FUNCTION_BLOCK ResetPlotter (* Composite Function Block Type *)
  (* Standard: 61499-2 *)
  (* Version 1.0, 2020-03-02, Mario *)
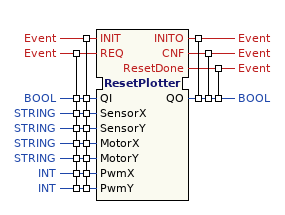
  EVENT_INPUT
    INIT WITH QI, SensorX, SensorY, MotorX, MotorY, PwmX, PwmY; (* Initialization Request *)
    REQ WITH QI, SensorX, SensorY, MotorX, MotorY, PwmX, PwmY; (* Normal Execution Request *)
  END_EVENT
  EVENT_OUTPUT
    INITO WITH QO; (* Initialization Confirm *)
    CNF WITH QO; (* Execution Confirmation *)
    ResetDone WITH QO;
  END_EVENT
  VAR_INPUT
    QI : BOOL; (* Input event qualifier *)
    SensorX : STRING;
    SensorY : STRING;
    MotorX : STRING;
    MotorY : STRING;
    PwmX : INT;
    PwmY : INT;
  END_VAR
  VAR_OUTPUT
    QO : BOOL; (* Output event qualifier *)
  END_VAR
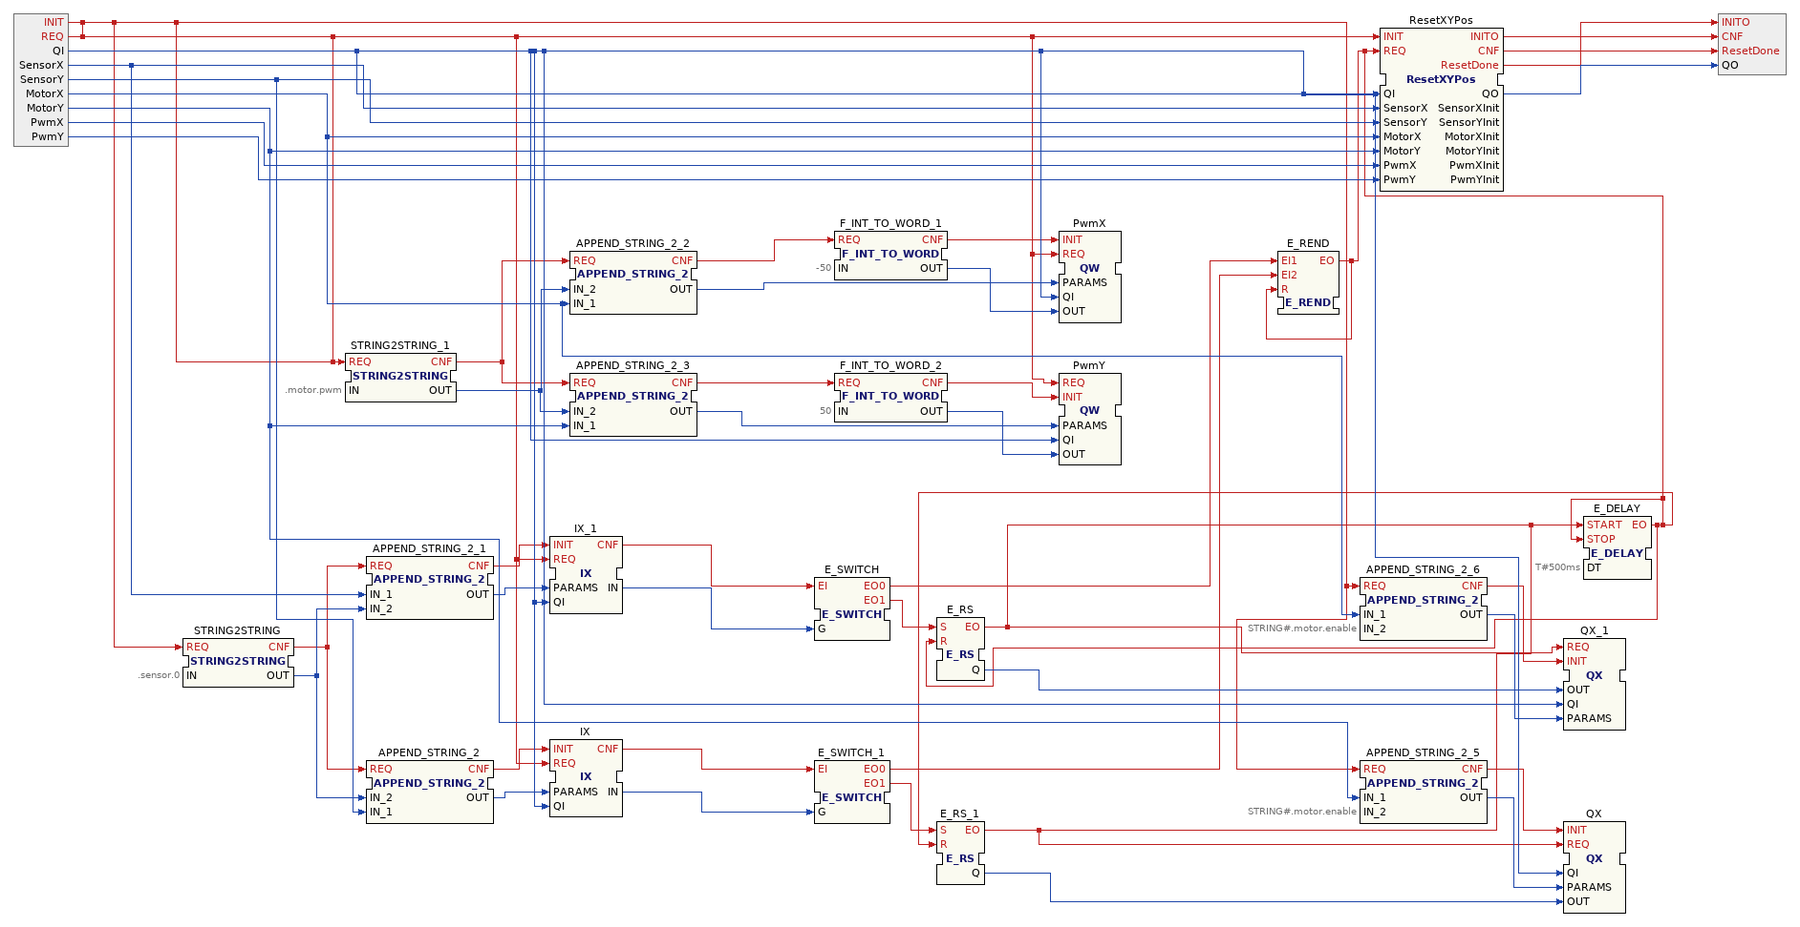
  FBS
    ResetXYPos : ResetXYPos;
    IX : IX;
    STRING2STRING : STRING2STRING(IN := .sensor.0);
    APPEND_STRING_2 : APPEND_STRING_2;
    IX_1 : IX;
    APPEND_STRING_2_1 : APPEND_STRING_2;
    E_SWITCH : E_SWITCH;
    E_SWITCH_1 : E_SWITCH;
    E_REND : E_REND;
    QX : QX;
    E_RS : E_RS;
    E_DELAY : E_DELAY(DT := T#500ms);
    PwmX : QW;
    PwmY : QW;
    STRING2STRING_1 : STRING2STRING(IN := .motor.pwm);
    APPEND_STRING_2_2 : APPEND_STRING_2;
    APPEND_STRING_2_3 : APPEND_STRING_2;
    QX_1 : QX;
    APPEND_STRING_2_5 : APPEND_STRING_2(IN_2 := STRING#.motor.enable);
    APPEND_STRING_2_6 : APPEND_STRING_2(IN_2 := STRING#.motor.enable);
    E_RS_1 : E_RS;
    F_INT_TO_WORD_1 : F_INT_TO_WORD(IN := -50);
    F_INT_TO_WORD_2 : F_INT_TO_WORD(IN := 50);
  END_FBS
  EVENT_CONNECTIONS
    INIT TO ResetXYPos.INIT;
    STRING2STRING.CNF TO APPEND_STRING_2_1.REQ;
    STRING2STRING.CNF TO APPEND_STRING_2.REQ;
    IX_1.CNF TO E_SWITCH.EI;
    IX.CNF TO E_SWITCH_1.EI;
    E_SWITCH.EO0 TO E_REND.EI1;
    E_SWITCH_1.EO0 TO E_REND.EI2;
    E_REND.EO TO E_REND.R;
    E_SWITCH.EO1 TO E_RS.S;
    E_RS.EO TO E_DELAY.START;
    E_DELAY.EO TO E_DELAY.STOP;
    E_DELAY.EO TO E_RS.R;
    STRING2STRING_1.CNF TO APPEND_STRING_2_2.REQ;
    STRING2STRING_1.CNF TO APPEND_STRING_2_3.REQ;
    INIT TO STRING2STRING_1.REQ;
    E_REND.EO TO ResetXYPos.REQ;
    ResetXYPos.ResetDone TO ResetDone;
    ResetXYPos.CNF TO CNF;
    ResetXYPos.INITO TO INITO;
    INIT TO STRING2STRING.REQ;
    APPEND_STRING_2_1.CNF TO IX_1.INIT;
    APPEND_STRING_2.CNF TO IX.INIT;
    REQ TO IX_1.REQ;
    REQ TO IX.REQ;
    REQ TO PwmY.REQ;
    E_RS.EO TO QX_1.REQ;
    INIT TO APPEND_STRING_2_6.REQ;
    INIT TO APPEND_STRING_2_5.REQ;
    APPEND_STRING_2_6.CNF TO QX_1.INIT;
    APPEND_STRING_2_5.CNF TO QX.INIT;
    E_SWITCH_1.EO1 TO E_RS_1.S;
    E_RS_1.EO TO QX.REQ;
    E_DELAY.EO TO E_RS_1.R;
    REQ TO STRING2STRING_1.REQ;
    E_DELAY.EO TO ResetXYPos.REQ;
    APPEND_STRING_2_2.CNF TO F_INT_TO_WORD_1.REQ;
    F_INT_TO_WORD_1.CNF TO PwmX.INIT;
    APPEND_STRING_2_3.CNF TO F_INT_TO_WORD_2.REQ;
    F_INT_TO_WORD_2.CNF TO PwmY.INIT;
    REQ TO PwmX.REQ;
    E_RS_1.EO TO E_DELAY.START;
  END_CONNECTIONS
  DATA_CONNECTIONS
    QI TO ResetXYPos.QI;
    SensorX TO ResetXYPos.SensorX;
    SensorY TO ResetXYPos.SensorY;
    MotorX TO ResetXYPos.MotorX;
    MotorY TO ResetXYPos.MotorY;
    PwmX TO ResetXYPos.PwmX;
    PwmY TO ResetXYPos.PwmY;
    STRING2STRING.OUT TO APPEND_STRING_2.IN_2;
    SensorX TO APPEND_STRING_2_1.IN_1;
    SensorY TO APPEND_STRING_2.IN_1;
    APPEND_STRING_2.OUT TO IX.PARAMS;
    APPEND_STRING_2_1.OUT TO IX_1.PARAMS;
    STRING2STRING.OUT TO APPEND_STRING_2_1.IN_2;
    IX_1.IN TO E_SWITCH.G;
    IX.IN TO E_SWITCH_1.G;
    QI TO IX_1.QI;
    QI TO IX.QI;
    STRING2STRING_1.OUT TO APPEND_STRING_2_3.IN_2;
    STRING2STRING_1.OUT TO APPEND_STRING_2_2.IN_2;
    MotorX TO APPEND_STRING_2_2.IN_1;
    MotorY TO APPEND_STRING_2_3.IN_1;
    APPEND_STRING_2_2.OUT TO PwmX.PARAMS;
    APPEND_STRING_2_3.OUT TO PwmY.PARAMS;
    ResetXYPos.QO TO QO;
    QI TO QX.QI;
    QI TO PwmX.QI;
    QI TO PwmY.QI;
    E_RS.Q TO QX_1.OUT;
    QI TO QX_1.QI;
    MotorX TO APPEND_STRING_2_6.IN_1;
    MotorY TO APPEND_STRING_2_5.IN_1;
    APPEND_STRING_2_6.OUT TO QX_1.PARAMS;
    APPEND_STRING_2_5.OUT TO QX.PARAMS;
    E_RS_1.Q TO QX.OUT;
    F_INT_TO_WORD_1.OUT TO PwmX.OUT;
    F_INT_TO_WORD_2.OUT TO PwmY.OUT;
  END_CONNECTIONS
END_FUNCTION_BLOCK
